ADAPTER ADPI_PRODUCTION_SERVICE (* Adapter Interface *)
  (* Standard: 61499-1 *)
  (* Version 0.0, 12/17/2022, Dmitrii, Flexbridge AB *)
  PACKAGE UAO.Hackathon;
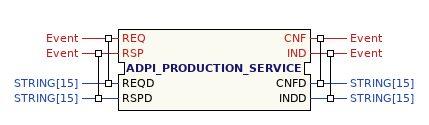
  EVENT_INPUT
    REQ WITH REQD; (* Request from Socket *)
    RSP WITH RSPD; (* Response from Socket *)
  END_EVENT
  EVENT_OUTPUT
    CNF WITH CNFD; (* Confirmation from Plug *)
    IND WITH INDD; (* Indication from Plug *)
  END_EVENT
  VAR_INPUT
    REQD : STRING[15]; (* Request Data from Socket *)
    RSPD : STRING[15]; (* Response Data from Socket *)
  END_VAR
  VAR_OUTPUT
    CNFD : STRING[15]; (* Confirmation Data from Plug *)
    INDD : STRING[15]; (* Indication Data from Plug *)
  END_VAR
  SERVICE SOCKET/PLUG
    SEQUENCE request_confirm
      SOCKET.REQ(REQD) -> PLUG.REQ(REQD);
      PLUG.CNF(CNFD) -> SOCKET.CNF(CNFD);
    END_SEQUENCE
    SEQUENCE indication_response
      PLUG.IND(INDD) -> SOCKET.IND(INDD);
      SOCKET.RSP(RSPD) -> PLUG.RSP(RSPD);
    END_SEQUENCE
  END_SERVICE
END_ADAPTER
